PROGRAM PRG_IO
VAR
	
	TextTimer: ton;
	Message_timer: ton;
	
	//List_of_Recipes				:ARRAY[1..10] OF Recipe;
	recipe_default				:recipe;
	Current_Recipe				:Recipe;
	//old_recipe					:Recipe;
	empty_recipe				:Recipe;
	current_recipe_no			:INT:=1;
	saveas_recipe_no			:INT;
	load_recipe_no				:INT;
	delete_recipe_no			:INT;
	temp						:INT;
	temp2						:INT;
		
	Initialise					:BOOL := TRUE;
	InitialiseTickCounter		:INT;
	TickCounter					:INT;
	
	save_requested				:BOOL := FALSE;
	
	Pusher_Home					:BOOL;
	Shield_Home					:BOOL;
	Compress_Home				:BOOL;
	
	//violation
	old_recipe					:Recipe;
	old_limits					:Limits;
	zero_violation				:BOOL;
	max_distance_violation		:BOOL;
	max_sh_push_diff_violation	:BOOL;
	
	Message_old					:STRING(300);
	
END_VAR

ResetLampController();
StartLampController();
TextTimer();
Message_timer();

//old_recipe:=current_recipe;

IF Initialise THEN
	InitialiseTickCounter := InitialiseTickCounter + 1;
	IF InitialiseTickCounter = 150 THEN
		Config.CopyConfigRecipiesToGlobal();
	END_IF		
	IF InitialiseTickCounter >= 300 THEN	
	//recipe_screen := List_of_Recipes[1];
		recipe_default.Name:='default 1';
	
		recipe_default.Compress.Initial_Distance:=60;
		recipe_default.Compress.Initial_Speed:=20;
		recipe_default.Compress.Relax_Distance:=5;
		recipe_default.Compress.Retract_Speed:=20;
	
		recipe_default.Pusher.Initial_Distance:=40;
		recipe_default.Pusher.Initial_Speed:=20;
		recipe_default.Pusher.Eject_Distance:=5;
		recipe_default.Pusher.Eject_Speed:=20;
		recipe_default.Pusher.Retract_Speed:=20;
	
		recipe_default.Shield.Retract_Speed:=20;
		recipe_default.Shield.Initial_Distance:=40;
		recipe_default.Shield.Initial_Speed:=20;
		
	
		recipe_default.Memory_Free:=FALSE;
	
		List_of_Recipes[1]:=recipe_default;
		recipe_screen:=List_of_Recipes[1];	
		
		limits_screen:=limits_save;
		
		Message:='Welcome!';
	
		InitialiseTickCounter := 0;
		Initialise := FALSE;
	END_IF		
ELSE
	InitialiseTickCounter := 0;

	current_recipe:=recipe_screen;

	//current_recipe_message:=CONCAT('The current recipe number is ',INT_TO_STRING(Current_recipe_no));
	
	IF current_recipe_no = 1 THEN
		Default_Recipe_Visibility:=FALSE;
	ELSE
		Default_Recipe_Visibility:=TRUE;
	END_IF
	
	FOR	temp := 1 TO 10 DO
		Recipe_Visibility[temp]:=NOT(List_of_Recipes[temp].Memory_Free);
	END_FOR
	
	temp:=1;
END_IF


//violation

IF  recipe_screen.Compress.Initial_Distance =0 OR 
	recipe_screen.Compress.Initial_Speed =0 OR 
	recipe_screen.Compress.Relax_Distance =0 OR 
	recipe_screen.Compress.Retract_Speed =0 OR
	recipe_screen.Pusher.Eject_Distance = 0 OR
	recipe_screen.pusher.Eject_Speed = 0 OR
	recipe_screen.pusher.Initial_Distance = 0 OR
	recipe_screen.Pusher.Initial_Speed = 0 OR
	recipe_screen.Pusher.Retract_Speed = 0 OR
	recipe_screen.Shield.Retract_Speed = 0 THEN
		
	zero_violation := TRUE;
		
	//Message:='Axis Parameters cannot be set to zero';
		
	//recipe_screen := old_recipe;
	//limits_screen := old_limits;
	
ELSE
	zero_violation := FALSE;
END_IF
	
IF 	recipe_screen.Compress.Initial_Distance + recipe_screen.Other.Compress_Home_Offset > limits_screen.max_limit_compress OR
	recipe_screen.Compress.Relax_Distance + recipe_screen.Other.Compress_Home_Offset > limits_screen.max_limit_compress OR
	recipe_screen.Shield.Initial_Distance + recipe_screen.Other.Shield_Home_Offset > limits_screen.max_limit_shield OR
	recipe_screen.Pusher.Initial_Distance + recipe_screen.Other.Pusher_Home_Offset > limits_screen.max_limit_Pusher OR
	recipe_screen.Pusher.tamp_initial_distance + recipe_screen.Other.Pusher_Home_Offset > limits_screen.max_limit_Pusher OR
	recipe_screen.Pusher.tamp_final_distance + recipe_screen.Other.Pusher_Home_Offset > limits_screen.max_limit_Pusher OR
	recipe_screen.Pusher.Eject_Distance + recipe_screen.Other.Pusher_Home_Offset > limits_screen.max_limit_Pusher THEN
		
	max_distance_violation:=TRUE;
		
	//Message:='Maximum Limit Violation';
		
	//recipe_screen := old_recipe;
	//limits_screen := old_limits;
		
ELSE
	max_distance_violation:=FALSE;
END_IF

IF 	(recipe_screen.Other.Pusher_Home_Offset) - (recipe_screen.Other.Shield_Home_Offset) > limits_screen.max_pusher_shield_diff OR
	(recipe_screen.Pusher.Initial_Distance + recipe_screen.Other.Pusher_Home_Offset) - (recipe_screen.Shield.Initial_Distance + recipe_screen.Other.Shield_Home_Offset) > limits_screen.max_pusher_shield_diff OR                      
	(recipe_screen.Pusher.tamp_initial_distance + recipe_screen.Other.Pusher_Home_Offset) - (0 + recipe_screen.Other.Shield_Home_Offset) > limits_screen.max_pusher_shield_diff OR
	(recipe_screen.Pusher.tamp_final_distance + recipe_screen.Other.Pusher_Home_Offset) - (0 + recipe_screen.Other.Shield_Home_Offset) > limits_screen.max_pusher_shield_diff OR
	(recipe_screen.Pusher.Eject_Distance + recipe_screen.Other.Pusher_Home_Offset) - (0 + recipe_screen.Other.Shield_Home_Offset) > limits_screen.max_pusher_shield_diff THEN          
		
	max_sh_push_diff_violation := TRUE;
	
	//Message:='Maximum pusher-shield distance difference violation';
	
	//recipe_screen := old_recipe;
	//limits_screen := old_limits;
		
ELSE
	max_sh_push_diff_violation:=FALSE;
END_IF

IF max_sh_push_diff_violation OR max_distance_violation OR zero_violation THEN
	parameter_violation:=TRUE;
ELSE
	parameter_violation:=FALSE;
END_IF

old_recipe:=recipe_screen;
old_limits:=limits_screen;
//violation end



//alarms
IF zero_violation THEN
	alarm_message:='Some parameters can not be set to zero.'; 
END_IF

IF max_distance_violation THEN
	alarm_message:='Maximum axis distance violation'; 
END_IF

IF max_sh_push_diff_violation THEN
	alarm_message:='Maximum pusher-shield distance difference violation';; 
END_IF

IF Clamp_Alarm THEN
	alarm_message:='Clamp Overtime';
END_IF

IF Overtorque_alarm THEN
	alarm_message:='Motor Overtorque';
END_IF

IF NOT ixGuardOkay THEN
	alarm_message:='Guard Open';
END_IF

IF NOT CabinetE_StopButtonOkay THEN
	alarm_message:='E-Stop Pressed';
END_IF

IF CabinetE_StopButtonOkay AND ixGuardOkay AND NOT parameter_violation AND NOT Overtorque_alarm AND NOT Clamp_Alarm THEN
	alarm_message:='';
END_IF
//end_of_alarms

//save as request
IF SaveasRecipe = TRUE THEN
	saveas_recipe_no:=current_recipe_no;
	WHILE (List_of_Recipes[saveas_recipe_no].Memory_Free = FALSE) AND (saveas_recipe_no<11) DO  
		saveas_recipe_no:=saveas_recipe_no+1;
		
	END_WHILE
	
	IF saveas_recipe_no > 10 THEN
		Message:='Maximum Recipe limit has been reached';
		saveas_recipe_no:=10;
		SaveasRecipe := FALSE;	
	END_IF
		
	IF List_of_Recipes[saveas_recipe_no].Memory_Free = TRUE THEN
		SaveasRecipe:=FALSE;
		
		Message := 'Adding new recipe...';

		List_of_Recipes[saveas_recipe_no]:=current_recipe;
		List_of_Recipes[saveas_recipe_no].Name:=Saveas_name;
		List_of_Recipes[saveas_recipe_no].Memory_Free:=FALSE;
		//current_recipe:=recipe_screen;
		//Config.CopyGlobalRecipiesToConfig();
		
		//Current_Recipe := List_of_Recipes[current_recipe_no];
		//recipe_screen:=current_recipe;

		save_requested := TRUE;		
	
	END_IF
	
END_IF
//save as request end

//load recipe
FOR temp := 1 TO 10 DO
	IF LoadRecipe[temp] = TRUE THEN
		load_recipe_no := temp;
		LoadRecipe[temp] := FALSE;
		
		question := CONCAT('Do you want to save recipe ', recipe_screen.Name);
		question := CONCAT(question,', before loading the recipe ');
		question := CONCAT(question, List_of_Recipes[load_recipe_no].Name);
		question := CONCAT(question,'?'); 
	END_IF
END_FOR

IF Load_Request = TRUE THEN
	
	Load_Request:=FALSE;
	
	IF(Save_before_load=TRUE)THEN
		
		//current_recipe:=recipe_screen;
		List_of_Recipes[current_recipe_no] := current_recipe;
		List_of_Recipes[current_recipe_no].Memory_Free := FALSE;
		//config.CopySettingsFromGlobal();
		Save_before_load := FALSE;
		
		Message := CONCAT('Recipe ',recipe_screen.Name);
		Message := CONCAT(Message,' saving... ');
		
		save_requested := TRUE;	
		
	END_IF
	
	current_recipe_no:=load_recipe_no;
		
	Current_Recipe := List_of_Recipes[current_recipe_no];
	recipe_screen:=current_recipe;
	//Message := CONCAT('Recipe ',current_recipe.Name);
	//Message := CONCAT(Message,' loading... ');

	
END_IF
//load recipe end

//delete recipe
FOR temp := 1 TO 10 DO
	IF DeleteRecipe[temp] = TRUE THEN
		delete_recipe_no := temp;
		DeleteRecipe[temp] := FALSE;
		
		question := CONCAT('Do you want to delete recipe ', List_of_Recipes[delete_recipe_no].Name);
		question := CONCAT(question,'?'); 
	END_IF
END_FOR

IF Delete_Request = TRUE THEN
	
	Delete_Request:=FALSE;
	
	current_recipe_no:=delete_recipe_no;
	
	Message := CONCAT('Recipe ',List_of_Recipes[current_recipe_no].Name );
	Message := CONCAT(Message,' deleting...');
	
	WHILE (delete_recipe_no<10) AND List_of_Recipes[delete_recipe_no+1].Memory_Free = FALSE DO
		List_of_Recipes[delete_recipe_no]:=List_of_Recipes[delete_recipe_no+1];
		delete_recipe_no:=delete_recipe_no+1;
	END_WHILE
	
	List_of_Recipes[delete_recipe_no] := empty_recipe;
	//List_of_Recipes[delete_recipe_no].Memory_Free:=FALSE;
	
	
	IF current_recipe_no = delete_recipe_no AND current_recipe_no <> 1 THEN
		current_recipe_no := current_recipe_no - 1;
	END_IF
		
	Current_Recipe := List_of_Recipes[current_recipe_no];
	recipe_screen:=current_recipe;
	
	save_requested := TRUE;

	
END_IF
//delete recipe end

//save recipe
IF SaveRecipe THEN
	SaveRecipe := FALSE;
	//current_recipe:=recipe_screen;
	//recipe_screen:=current_recipe;
	current_recipe.Memory_Free:=FALSE;
	
	//WHILE (List_of_Recipes[current_recipe_no].Memory_Free = FALSE) AND (current_recipe_no<11) DO  
	//	current_recipe_no:=current_recipe_no+1;
	//END_WHILE
	Message := 'Recipe saving...';	
	
	List_of_Recipes[current_recipe_no] := current_recipe;
	save_requested := TRUE;
	
END_IF
//save recipe end

//save limits
IF save_limits THEN
	save_limits:=FALSE;
	limits_save:=limits_screen;
	save_requested := TRUE;
	Message:='Saving Limits...';
END_IF



IF save_requested = TRUE THEN
	
	save_requested := FALSE;
	Config.CopyGlobalRecipiesToConfig();
	config_request:= TRUE;
	//config_count:=0;
	//Message:='Configuring...';
	
END_IF

//Message Timer
IF Message <> message_old THEN
	Message_timer.IN:=TRUE;
	Message_Timer.PT:=T#10S;
END_IF

IF Message_Timer.Q = TRUE THEN
	Message:='';
	Message_timer.IN:=FALSE;
	//Message_Timer.PT:=T#30S;
END_IF 
Message_old:=Message;
//end of message timer


//Config.CopyGlobalRecipiesToConfig();
//end recipes


(***************************** Data For the Main Screen ***********************)


	(* Settings Page*)


	(* IO Page *)

CabinetE_StopButtonOkay := ixCabinetE_StopButtonOkay;
E_StopRelayOkay:=ixE_StopRelayOkay;
GuardRelayOkay:=ixGuardRelayOkay;
GuardOkay:=ixGuardOkay;

ResetButton := ixResetButton;

		
// Cabinet Digital Outputs 1 - Device 1, Term 3
EnableE_Stop:=qxEnableE_Stop;
	
//StartButtonLamp:=qxStartButtonLamp;
ResetButtonLamp:=qxResetButtonLamp;
	
	
// Servo Analogue Inputs 1- Device 2, Term 2
CompressServoTorque:=ibCompressServoTorque;
CompressServoFollowingError:=ibCompressServoFollowingError;
CompressServoTorqueLimit:=qbCompressServoTorqueLimit;
	
// Servo Analogue Inputs 1- Device 2, Term 3
PusherServoTorque:=ibPusherServoTorque;
PusherServoFollowingError:=ibPusherServoFollowingError;
PusherServoTorqueLimit:=qbPusherServoTorqueLimit;
	
// Servo Analogue Inputs 1- Device 2, Term 3
ShieldServoTorque:=ibShieldServoTorque;
ShieldServoFollowingError:=ibShieldServoFollowingError;
ShieldServoTorqueLimit:=qbShieldServoTorqueLimit;
	

	
// Machine Digital Inputs 1 - Device 2, Term 5
CompressHomeSwitch:=ixCompressHomeSwitch;
PusherHomeSwitch:=ixPusherHomeSwitch;
ShieldHomeSwitch:=ixShieldHomeSwitch;
StartButton:=ixStartButton;
GuardOkay:=ixGuardOkay; 
MachineE_StopButtonOkay:=ixMachineE_StopButtonOkay;
//FanCartridgeDiagnostics:=ixFanCartridgeDiagnostics;

//sc_CompressServoErrorID := CompressServoErrorID;
//sc_PusherServoErrorID := PusherServoErrorID;	
//sc_ShieldServoErrorID := ShieldServoErrorID;
	

//Homed?
Pusher_Home:=PRG_Machine.Pusher.HomeExecuted;
Shield_Home:=PRG_Machine.Shield.HomeExecuted;
Compress_Home:=PRG_Machine.Compress.HomeExecuted;
	
//Clamp
Clamp_State:=qxClamp;

//Mode
IF debug_mode = FALSE THEN
	mode_string:= 'Current Mode: Automatic';
ELSE
	mode_string:= 'Current Mode: Debug';
END_IF

//until here





qxResetButtonLamp := ResetLampController.Q; //io
ResetLamp := ResetLampController.Q; //zenon



ShieldAxisPosition := PRG_Machine.Shield.ShieldServo.fActualPosition;		
PusherAxisPosition := PRG_Machine.Pusher.PusherServo.fActualPosition;
CompressAxisPosition := PRG_Machine.Compress.CompressServo.fActualPosition;

Zenon_Offset_Compress:=PRG_Machine.Compress.OffsetExecuted;
Zenon_Offset_Shield:=PRG_Machine.Shield.OffsetExecuted;
Zenon_Offset_Pusher:=PRG_Machine.Pusher.OffsetExecuted;
		
	(* Top Bar *)
//	sSystemState			: STRING;		//Top Bar
(*		
IF sSystemStateHi = WSTRING_TO_STRING("") THEN
	IF sSystemStateMed = WSTRING_TO_STRING("") THEN
		sSystemState := sSystemStateLo;
	ELSE
		sSystemState := sSystemStateMed;
	END_IF	
ELSE
	sSystemState := sSystemStateHi;
	TextTimer.PT := T#5S;
	TextTimer.IN := TRUE;
	IF TextTimer.Q THEN
		sSystemStateHi :=  WSTRING_TO_STRING("");
		TextTimer.IN := false;
	END_IF
END_IF

sc_sSystemStateHi := sSystemStateHi;
sc_sSystemStateMed := sSystemStateMed;
sc_sSystemStateLo := sSystemStateLo;

*)

PROPERTY List_of_Recipes_config :ARRAY[1..10] OF Recipe;
GET
List_of_Recipes_config := List_of_Recipes;
END_GET
SET
List_of_Recipes := List_of_Recipes_config;
END_SET
END_PROPERTY

PROPERTY recipe_default_ext :Recipe;
GET
recipe_default_ext := recipe_default;
END_GET
SET
recipe_default := recipe_default_ext;
END_SET
END_PROPERTY

END_PROGRAM

(* stored: Version 1.1.0.1, ProductVersion 3.1.4020.12
   POU PRG_IO: Id {f101afa0-f9ee-4197-8bc4-4b48547efe33}, SpecialFunc None
   Property List_of_Recipes_config: Id {92324b27-23cd-4b80-9414-75de92c10226}
   Get Get: Id {f93cf17d-52c3-4715-a269-8274f1b057d6}
   Set Set: Id {29a903ab-de62-4fef-8203-1ec5ccafa9c7}
   Property recipe_default_ext: Id {004faa73-251f-4e55-9276-5e6e11f50fae}
   Get Get: Id {077e0aaa-22a5-4b34-be0f-cbc181a1f8ae}
   Set Set: Id {55dbf694-5b08-4539-9a9e-f402110f2108} *)
